{attribute addProperty BoxType "IODEVICETYPE_ETHERCATPROT"}
{attribute addProperty Id "Beckhoff_AT1xxxBeckhoff_AT1xxx_734BE41E471205890Beckhoff_ATH2xxxBeckhoff_ATH2xxx_4821DE8E7072884SyncUnitsSyncUnits_3FA29F3C21627InputsInputs_C75D3FEC1280160OutputsOutputs_47D1E803848106InfoDataInfoData_45F98C5022428"}
{attribute addProperty CRC "2626821938"}
{attribute addProperty SizeInBites "56760"}
{attribute addProperty SizeInBytes "7095"}
TYPE EtherCAT_Master_ATxxxx_9C921F32 :
STRUCT
	{attribute addProperty Name "Beckhoff_AT1xxx"}
	Beckhoff_AT1xxx : Beckhoff_AT1xxx_734BE41E;
	{attribute addProperty Name "Beckhoff_ATH2xxx"}
	Beckhoff_ATH2xxx : Beckhoff_ATH2xxx_4821DE8E;
	{attribute addProperty Name "SyncUnits"}
	SyncUnits : SyncUnits_3FA29F3C;
	{attribute addProperty Name "Inputs"}
	Inputs : Inputs_C75D3FEC;
	{attribute addProperty Name "Outputs"}
	Outputs : Outputs_47D1E803;
	{attribute addProperty Name "InfoData"}
	InfoData : InfoData_45F98C50;
END_STRUCT
END_TYPE

(* stored: Version 1.2.0.0, ProductVersion 3.1.4024.9
   DUT EtherCAT_Master_ATxxxx_9C921F32: Id {ff92dd10-7184-46e8-a8c1-8de1db083c02} *)
